FUNCTION_BLOCK OpcUaCreatePaths (* Basic FB with empty ECC *)
  (* Standard: 61499-2; Description: Copyright (c) 2026 Monika Wenger This program and the accompanying materials are made available under the terms of the Eclipse Public License 2.0 which is available at https://www.eclipse.org/legal/epl-2.0/ SPDX-License-Identifier: EPL-2.0 *)
  (* Version 3.0, 2025-12-05, Monika Wenger *)
  PACKAGE eclipse4diac::opcua;
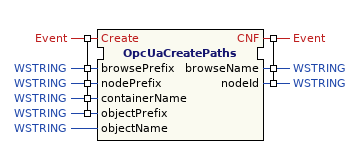
  EVENT_INPUT
    Create WITH containerName, browsePrefix, nodePrefix, objectPrefix;
  END_EVENT
  EVENT_OUTPUT
    CNF WITH browseName, nodeId;
  END_EVENT
  VAR_INPUT
    browsePrefix : WSTRING := "/Objects/skills/";
    nodePrefix : WSTRING := "skills.";
    containerName : WSTRING;
    objectPrefix : WSTRING;
    objectName : WSTRING;
  END_VAR
  VAR_OUTPUT
    browseName : WSTRING;
    nodeId : WSTRING;
  END_VAR
  VAR CONSTANT
    BROWSE_SEPARATOR : WSTRING := "/";
    NODE_SEPARATOR : WSTRING := ".";
  END_VAR
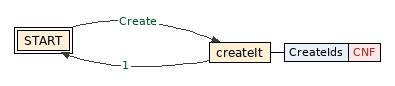
  EC_STATES
    START; (* Initial State *)
    createIt : CreateIds -> CNF;
  END_STATES
  EC_TRANSITIONS
    START TO createIt := Create;
    createIt TO START := 1;
  END_TRANSITIONS
  ALGORITHM CreateIds IN ST:
IF EQ(objectPrefix, "") THEN
	browseName := CONCAT(browsePrefix, containerName, BROWSE_SEPARATOR, objectName);
	nodeId := CONCAT(nodePrefix, containerName, NODE_SEPARATOR, objectName);
ELSE
	browseName := CONCAT(browsePrefix, containerName, BROWSE_SEPARATOR, objectPrefix, BROWSE_SEPARATOR, objectName);
	nodeId := CONCAT(nodePrefix, containerName, NODE_SEPARATOR, objectPrefix, NODE_SEPARATOR, objectName);
END_IF;
  END_ALGORITHM
END_FUNCTION_BLOCK
